DATA_BLOCK "CAROUSEL1"

{ S7_Optimized_Access := 'TRUE' }
VERSION : 0.1
NON_RETAIN
"Carousel_SEW_MOVIGEAR"

BEGIN

END_DATA_BLOCK
